PROGRAM main
VAR
	LocalStart AT %IX0.0 : bool;
	RemoteStart AT %IX0.1 : bool;
	MotorRun AT %QX0.0 : bool;
END_VAR

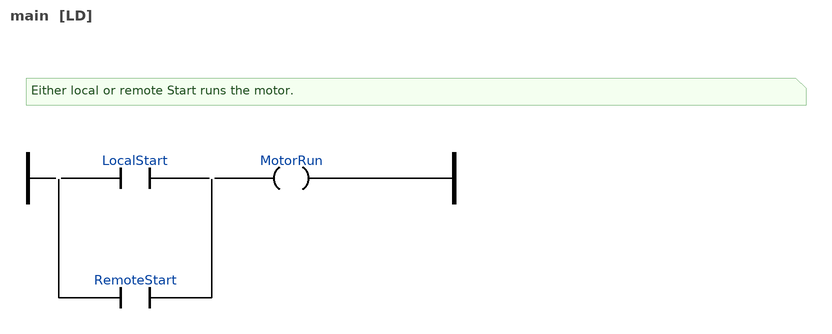
(* LD diagram, written out as Structured Text *)
(* Either local or remote Start runs the motor. *)
MotorRun := LocalStart OR RemoteStart;
END_PROGRAM
